Omron CX-Programmer project NewProject (CX-Programmer 9.73)

# PLC NewPLC1: CP2E-N N

## Global symbols (name address type ; comment)
0.00 BOOL  ; SW_ON
100.00 BOOL  ; LAMP 1
100.01 BOOL  ; LAMP 2
D0 CHANNEL  ; Error_Code
D20 CHANNEL  ; IP_Octet 1
D21 CHANNEL  ; IP_Octet 2
D22 CHANNEL  ; IP_Octet 3
D23 CHANNEL  ; IP_Octet 4
D24 CHANNEL  ; Port_Number
D9000 CHANNEL  ; Cut_Com
T000 BOOL  ; T_StartMODTCP
W0.00 BOOL  ; Server_Start_Flag
W1.01 BOOL  ; Error_Flag
ModbusTCP_IP _CP2E003_ExecuteModTcpServer

## Program NewProgram1 (cyclic task 0)

### Section Section1

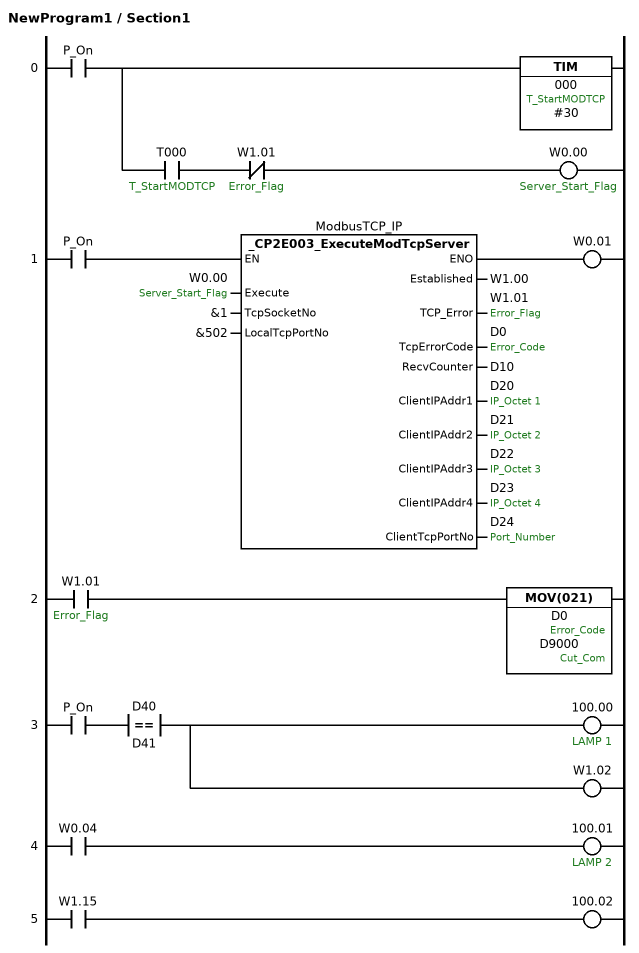
; rung 0
LD P_On
TIM 000 #30  ; T_StartMODTCP
AND T000  ; T_StartMODTCP
ANDNOT W1.01  ; Error_Flag
OUT W0.00  ; Server_Start_Flag
; rung 1
LD P_On
CALL ModbusTCP_IP : _CP2E003_ExecuteModTcpServer (Execute := W0.00, TcpSocketNo := &1, LocalTcpPortNo := &502, Established => W1.00, TCP_Error => W1.01, TcpErrorCode => D0, RecvCounter => D10, ClientIPAddr1 => D20, ClientIPAddr2 => D21, ClientIPAddr3 => D22, ClientIPAddr4 => D23, ClientTcpPortNo => D24)  ; Server_Start_Flag, Error_Flag, Error_Code, IP_Octet 1, IP_Octet 2, IP_Octet 3, IP_Octet 4, Port_Number
OUT W0.01
; rung 2
LD W1.01  ; Error_Flag
MOV(021) D0 D9000  ; Error_Code, Cut_Com
; rung 3
LD P_On
AND=(300) D40 D41
OUT 100.00  ; LAMP 1
OUT W1.02
; rung 4
LD W0.04
OUT 100.01  ; LAMP 2
; rung 5
LD W1.15
OUT 100.02

### Section END
; rung 0
END(001)

## Function block _CP2E003_ExecuteModTcpServer (Omron library block, body left out)